(* Logix 5000 project; controller cal1632 1756-L62 rev 16.20; software revision 16.05; part 28 of 61 *)
(* tags used below, declared in another part *)
   FAULT : BOOL;
   HMI : BOOL;
   p01_recipe_active : recipe;
   p01r09_pb_global_reset : BOOL;
   p02_dint_from_hmi : hmi_dint;
   p02_real_from_hmi : hmi_real;
   p20_ai_lc01 : REAL;
   p20_di_clutch_prs_ok : BOOL;
   p20_di_loa_active : BOOL;
   p20_di_loa_fwd_dir : BOOL;
   p20_di_lob_fwd_dir : BOOL;
   p20_dint_to_hmi : DINT[16];
   p20_param_high_ki : REAL;
   p20_param_high_kp : REAL;
   p20_param_high_upd : REAL;
   p20r07 : routine;
   p20r07_timer_fault : TIMER[4];
   p20r07_timer_warning : TIMER[4];
   p20r08 : routine;
   p20r08_timer_fault : TIMER[4];
   p20r08_timer_warning : TIMER[4];
   p20r09 : routine;
   p20r09_acc_toggle : SYS_Toggle;
   p20r09_accumulator_auto : BOOL;
   p20r09_letoff_a_active : BOOL;
   p20r09_timer_fault : TIMER[4];
   p20r09_timer_warning : TIMER[4];
   p20r10 : routine;
   p20r10_param_acc_full_psn : REAL;
   p20r10_param_fill_gain : REAL;
   p20r10_param_normal_gain : REAL;
   p20r10_param_psn_gain : REAL;
   p20r10_pid_psn : PID;
   p20r10_pid_psn_cv : REAL;
   p20r10_pid_psn_pv : REAL;
   p20r10_pid_tens : PID;
   p20r10_pid_tens_cv : REAL;
   p20r10_pid_tens_pv : REAL;
   p20r10_run_permissive : BOOL;
   p20r10_speed_offset : REAL;
   p20r10_speed_offset_psn : REAL;
   p20r10_speed_offset_tens : REAL;
   p20r10_tension_request : BOOL;
   p20r10_timer : TIMER[2];
   p20r10_timer_fault : TIMER[4];
   p20r10_timer_warning : TIMER[4];
   p20r13_ai_acc_pct : REAL;
   p20r13_state : DINT;
   p20r15 : routine;
   p20r15_request_tension : BOOL;
   p20r15_request_thread_fwd : BOOL;
   p20r15_request_thread_rev : BOOL;
   p20r16 : routine;
   p20r16_request_tension : BOOL;
   p20r16_request_thread_fwd : BOOL;
   p20r16_request_thread_rev : BOOL;
   p20r18 : routine;
(* P20_Letoff, continued *)

ROUTINE R07_Alarms   (* ladder *)
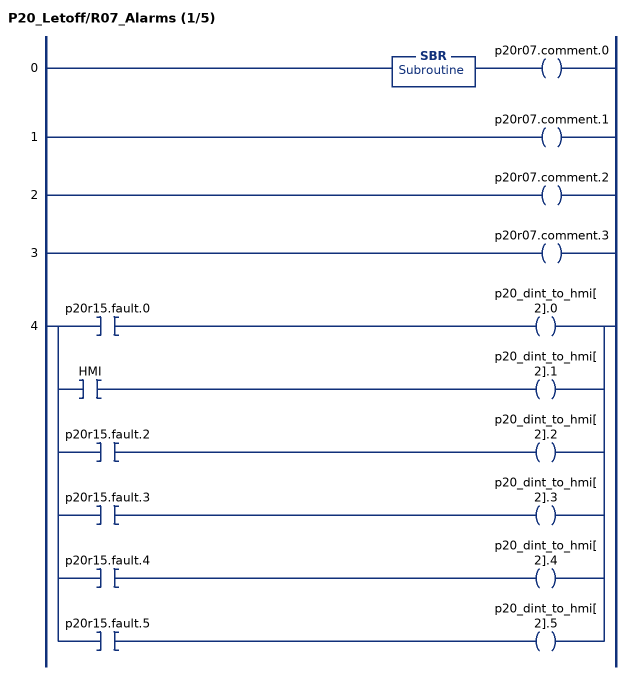
   0: SBR()OTE(p20r07.comment.0);
   1: OTE(p20r07.comment.1);
   2: OTE(p20r07.comment.2);
   3: OTE(p20r07.comment.3);
   4: [XIC(p20r15.fault.0) OTE(p20_dint_to_hmi[2].0) ,XIC(HMI) OTE(p20_dint_to_hmi[2].1) ,XIC(p20r15.fault.2) OTE(p20_dint_to_hmi[2].2) ,XIC(p20r15.fault.3) OTE(p20_dint_to_hmi[2].3) ,XIC(p20r15.fault.4) OTE(p20_dint_to_hmi[2].4) ,XIC(p20r15.fault.5) OTE(p20_dint_to_hmi[2].5) ];
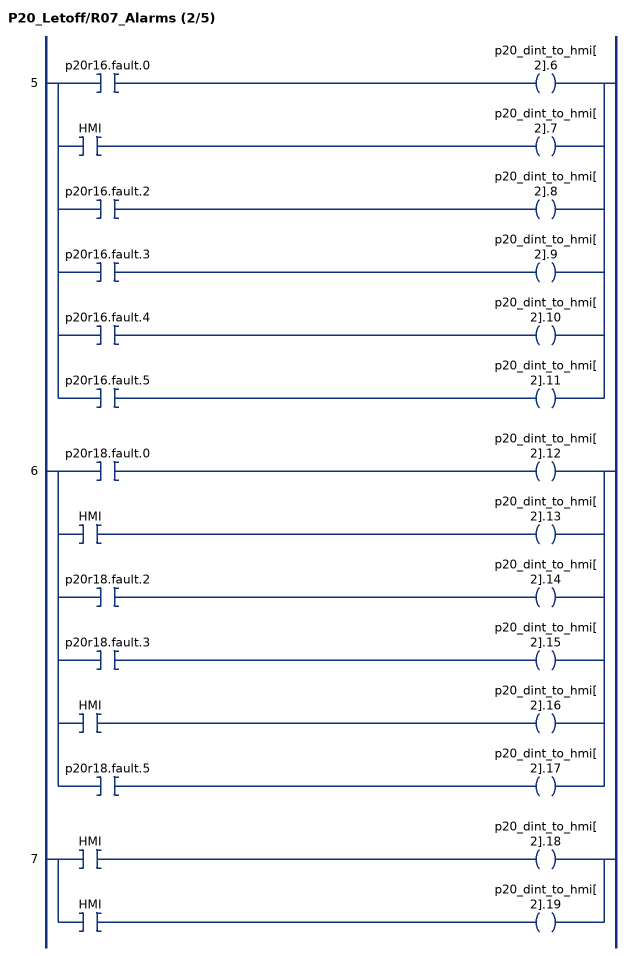
   5: [XIC(p20r16.fault.0) OTE(p20_dint_to_hmi[2].6) ,XIC(HMI) OTE(p20_dint_to_hmi[2].7) ,XIC(p20r16.fault.2) OTE(p20_dint_to_hmi[2].8) ,XIC(p20r16.fault.3) OTE(p20_dint_to_hmi[2].9) ,XIC(p20r16.fault.4) OTE(p20_dint_to_hmi[2].10) ,XIC(p20r16.fault.5) OTE(p20_dint_to_hmi[2].11) ];
   6: [XIC(p20r18.fault.0) OTE(p20_dint_to_hmi[2].12) ,XIC(HMI) OTE(p20_dint_to_hmi[2].13) ,XIC(p20r18.fault.2) OTE(p20_dint_to_hmi[2].14) ,XIC(p20r18.fault.3) OTE(p20_dint_to_hmi[2].15) ,XIC(HMI) OTE(p20_dint_to_hmi[2].16) ,XIC(p20r18.fault.5) OTE(p20_dint_to_hmi[2].17) ];
   7: [XIC(HMI) OTE(p20_dint_to_hmi[2].18) ,XIC(HMI) OTE(p20_dint_to_hmi[2].19) ];
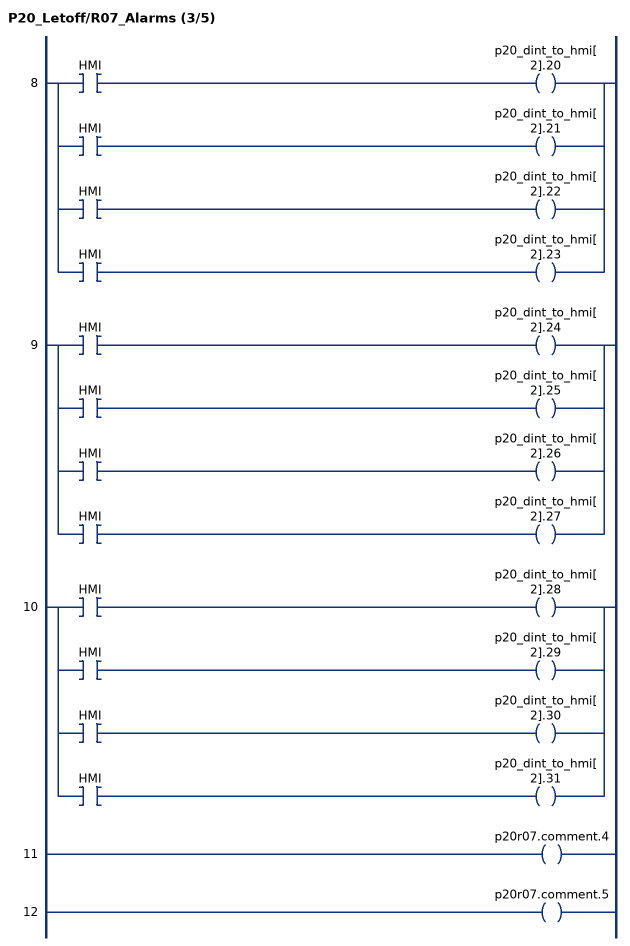
   8: [XIC(HMI) OTE(p20_dint_to_hmi[2].20) ,XIC(HMI) OTE(p20_dint_to_hmi[2].21) ,XIC(HMI) OTE(p20_dint_to_hmi[2].22) ,XIC(HMI) OTE(p20_dint_to_hmi[2].23) ];
   9: [XIC(HMI) OTE(p20_dint_to_hmi[2].24) ,XIC(HMI) OTE(p20_dint_to_hmi[2].25) ,XIC(HMI) OTE(p20_dint_to_hmi[2].26) ,XIC(HMI) OTE(p20_dint_to_hmi[2].27) ];
   10: [XIC(HMI) OTE(p20_dint_to_hmi[2].28) ,XIC(HMI) OTE(p20_dint_to_hmi[2].29) ,XIC(HMI) OTE(p20_dint_to_hmi[2].30) ,XIC(HMI) OTE(p20_dint_to_hmi[2].31) ];
   11: OTE(p20r07.comment.4);
   12: OTE(p20r07.comment.5);
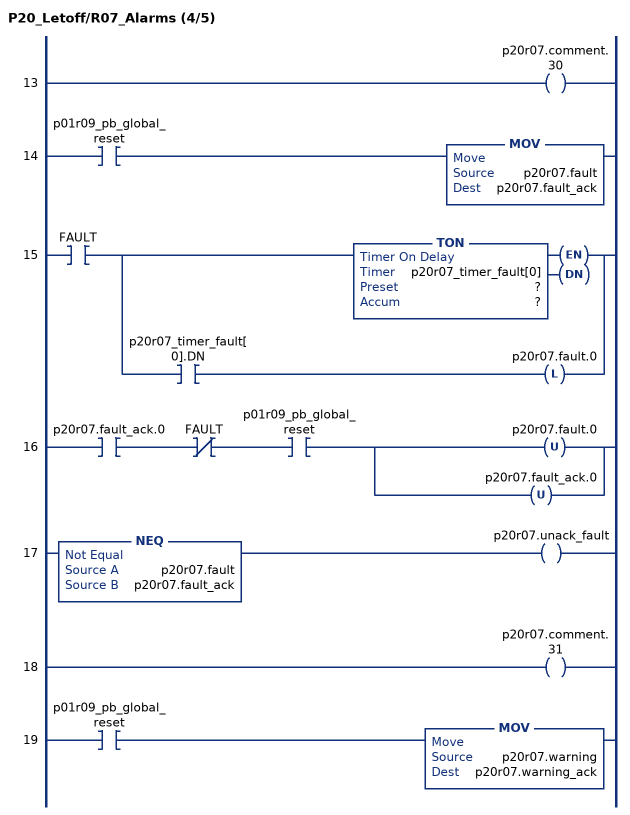
   13: OTE(p20r07.comment.30);
   14: XIC(p01r09_pb_global_reset)MOV(p20r07.fault,p20r07.fault_ack);
   15: XIC(FAULT)[TON(p20r07_timer_fault[0],?,?) ,XIC(p20r07_timer_fault[0].DN) OTL(p20r07.fault.0) ];
   16: XIC(p20r07.fault_ack.0)XIO(FAULT)XIC(p01r09_pb_global_reset)[OTU(p20r07.fault.0) ,OTU(p20r07.fault_ack.0) ];
   17: NEQ(p20r07.fault,p20r07.fault_ack)OTE(p20r07.unack_fault);
   18: OTE(p20r07.comment.31);
   19: XIC(p01r09_pb_global_reset)MOV(p20r07.warning,p20r07.warning_ack);
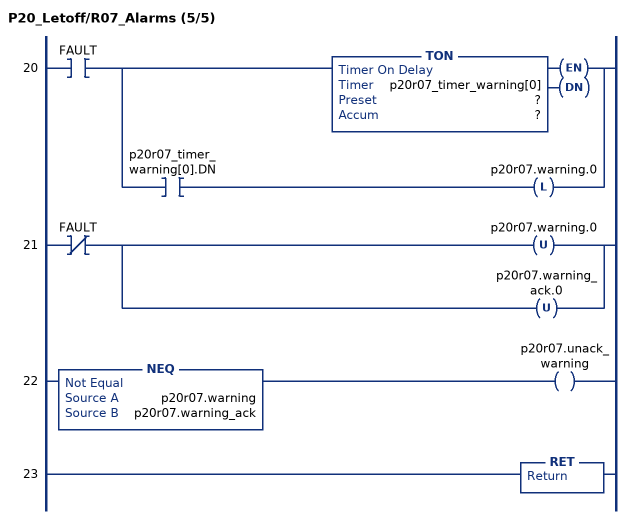
   20: XIC(FAULT)[TON(p20r07_timer_warning[0],?,?) ,XIC(p20r07_timer_warning[0].DN) OTL(p20r07.warning.0) ];
   21: XIO(FAULT)[OTU(p20r07.warning.0) ,OTU(p20r07.warning_ack.0) ];
   22: NEQ(p20r07.warning,p20r07.warning_ack)OTE(p20r07.unack_warning);
   23: RET();
END_ROUTINE

ROUTINE R08_Warnings   (* ladder *)
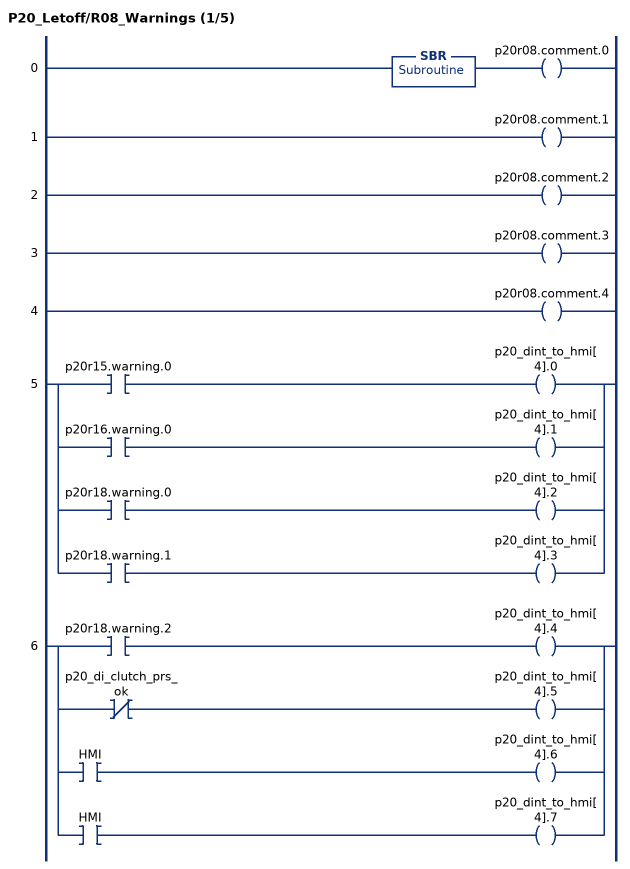
   0: SBR()OTE(p20r08.comment.0);
   1: OTE(p20r08.comment.1);
   2: OTE(p20r08.comment.2);
   3: OTE(p20r08.comment.3);
   4: OTE(p20r08.comment.4);
   5: [XIC(p20r15.warning.0) OTE(p20_dint_to_hmi[4].0) ,XIC(p20r16.warning.0) OTE(p20_dint_to_hmi[4].1) ,XIC(p20r18.warning.0) OTE(p20_dint_to_hmi[4].2) ,XIC(p20r18.warning.1) OTE(p20_dint_to_hmi[4].3) ];
   6: [XIC(p20r18.warning.2) OTE(p20_dint_to_hmi[4].4) ,XIO(p20_di_clutch_prs_ok) OTE(p20_dint_to_hmi[4].5) ,XIC(HMI) OTE(p20_dint_to_hmi[4].6) ,XIC(HMI) OTE(p20_dint_to_hmi[4].7) ];
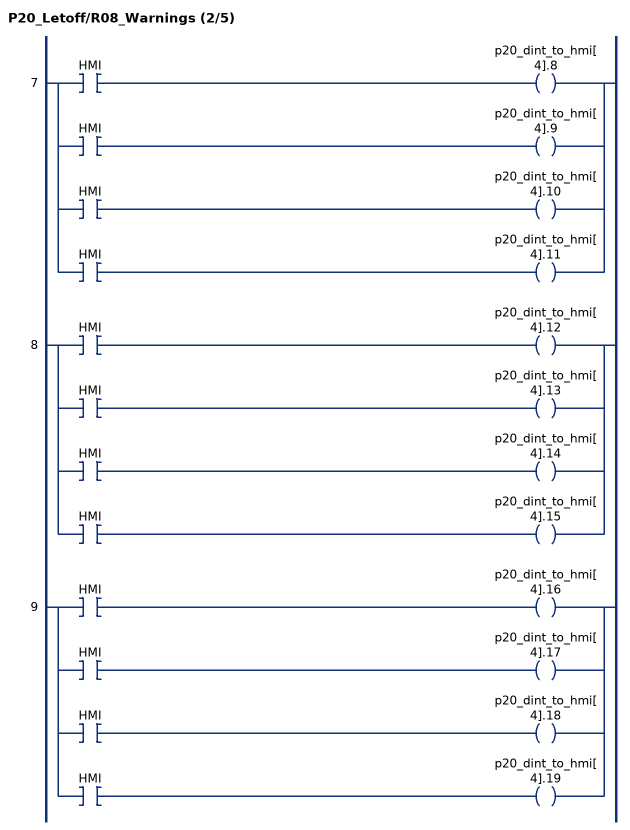
   7: [XIC(HMI) OTE(p20_dint_to_hmi[4].8) ,XIC(HMI) OTE(p20_dint_to_hmi[4].9) ,XIC(HMI) OTE(p20_dint_to_hmi[4].10) ,XIC(HMI) OTE(p20_dint_to_hmi[4].11) ];
   8: [XIC(HMI) OTE(p20_dint_to_hmi[4].12) ,XIC(HMI) OTE(p20_dint_to_hmi[4].13) ,XIC(HMI) OTE(p20_dint_to_hmi[4].14) ,XIC(HMI) OTE(p20_dint_to_hmi[4].15) ];
   9: [XIC(HMI) OTE(p20_dint_to_hmi[4].16) ,XIC(HMI) OTE(p20_dint_to_hmi[4].17) ,XIC(HMI) OTE(p20_dint_to_hmi[4].18) ,XIC(HMI) OTE(p20_dint_to_hmi[4].19) ];
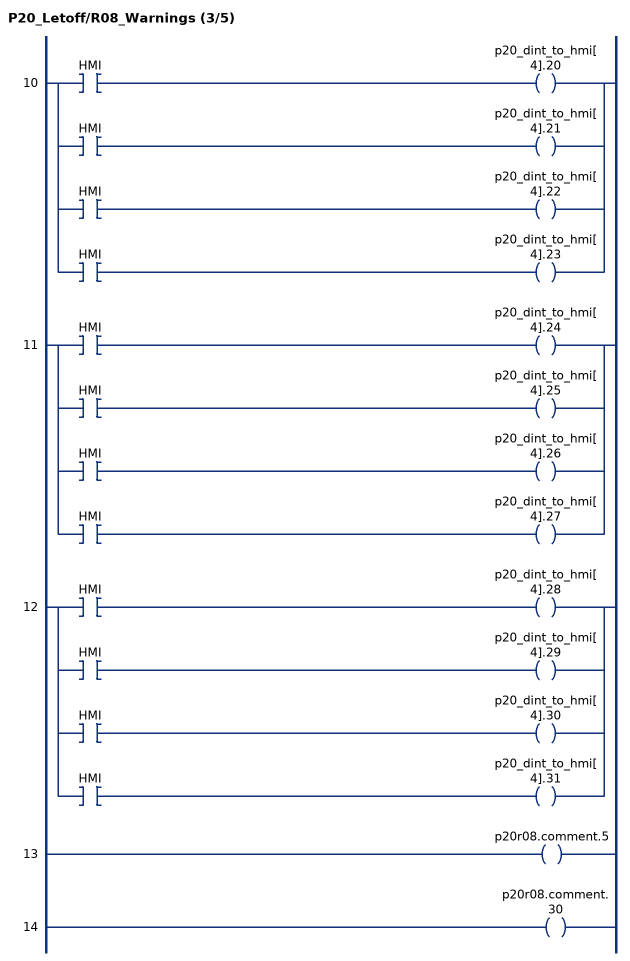
   10: [XIC(HMI) OTE(p20_dint_to_hmi[4].20) ,XIC(HMI) OTE(p20_dint_to_hmi[4].21) ,XIC(HMI) OTE(p20_dint_to_hmi[4].22) ,XIC(HMI) OTE(p20_dint_to_hmi[4].23) ];
   11: [XIC(HMI) OTE(p20_dint_to_hmi[4].24) ,XIC(HMI) OTE(p20_dint_to_hmi[4].25) ,XIC(HMI) OTE(p20_dint_to_hmi[4].26) ,XIC(HMI) OTE(p20_dint_to_hmi[4].27) ];
   12: [XIC(HMI) OTE(p20_dint_to_hmi[4].28) ,XIC(HMI) OTE(p20_dint_to_hmi[4].29) ,XIC(HMI) OTE(p20_dint_to_hmi[4].30) ,XIC(HMI) OTE(p20_dint_to_hmi[4].31) ];
   13: OTE(p20r08.comment.5);
   14: OTE(p20r08.comment.30);
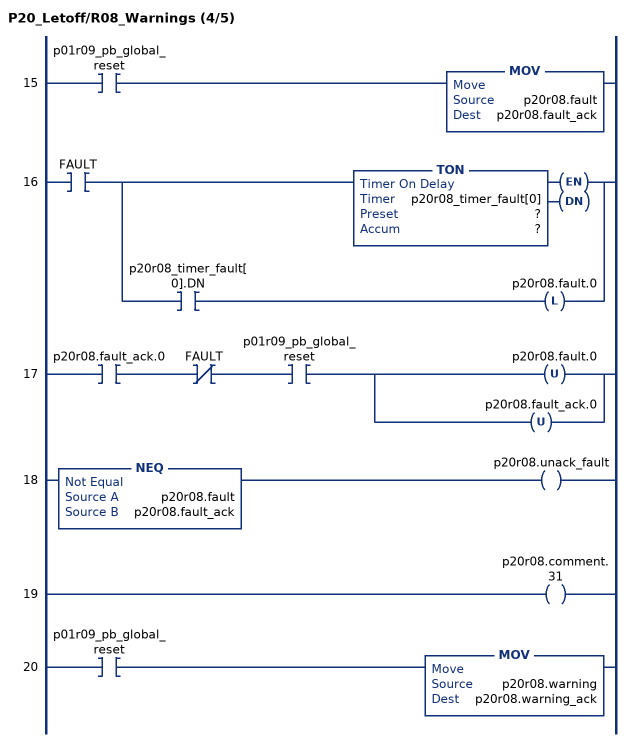
   15: XIC(p01r09_pb_global_reset)MOV(p20r08.fault,p20r08.fault_ack);
   16: XIC(FAULT)[TON(p20r08_timer_fault[0],?,?) ,XIC(p20r08_timer_fault[0].DN) OTL(p20r08.fault.0) ];
   17: XIC(p20r08.fault_ack.0)XIO(FAULT)XIC(p01r09_pb_global_reset)[OTU(p20r08.fault.0) ,OTU(p20r08.fault_ack.0) ];
   18: NEQ(p20r08.fault,p20r08.fault_ack)OTE(p20r08.unack_fault);
   19: OTE(p20r08.comment.31);
   20: XIC(p01r09_pb_global_reset)MOV(p20r08.warning,p20r08.warning_ack);
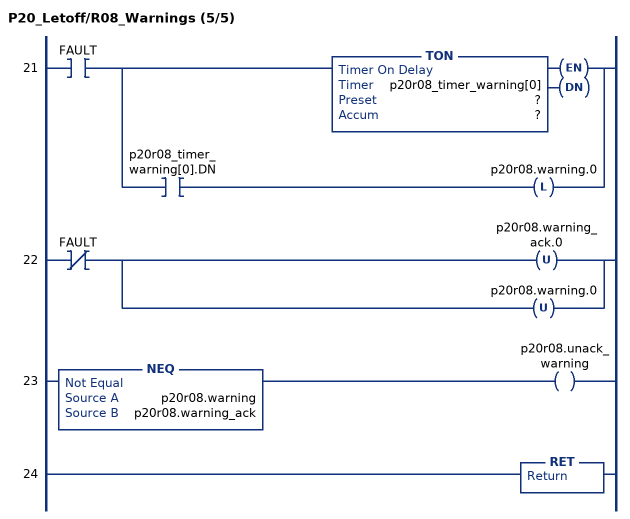
   21: XIC(FAULT)[TON(p20r08_timer_warning[0],?,?) ,XIC(p20r08_timer_warning[0].DN) OTL(p20r08.warning.0) ];
   22: XIO(FAULT)[OTU(p20r08.warning_ack.0) ,OTU(p20r08.warning.0) ];
   23: NEQ(p20r08.warning,p20r08.warning_ack)OTE(p20r08.unack_warning);
   24: RET();
END_ROUTINE

ROUTINE R09_Modes   (* ladder *)
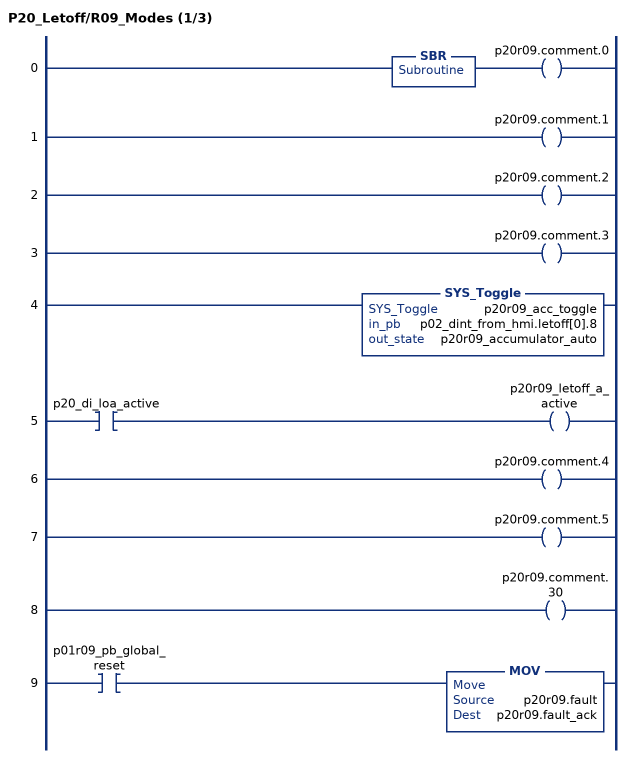
   0: SBR()OTE(p20r09.comment.0);
   1: OTE(p20r09.comment.1);
   2: OTE(p20r09.comment.2);
   3: OTE(p20r09.comment.3);
   4: SYS_Toggle(p20r09_acc_toggle,p02_dint_from_hmi.letoff[0].8,p20r09_accumulator_auto);
   5: XIC(p20_di_loa_active)OTE(p20r09_letoff_a_active);
   6: OTE(p20r09.comment.4);
   7: OTE(p20r09.comment.5);
   8: OTE(p20r09.comment.30);
   9: XIC(p01r09_pb_global_reset)MOV(p20r09.fault,p20r09.fault_ack);
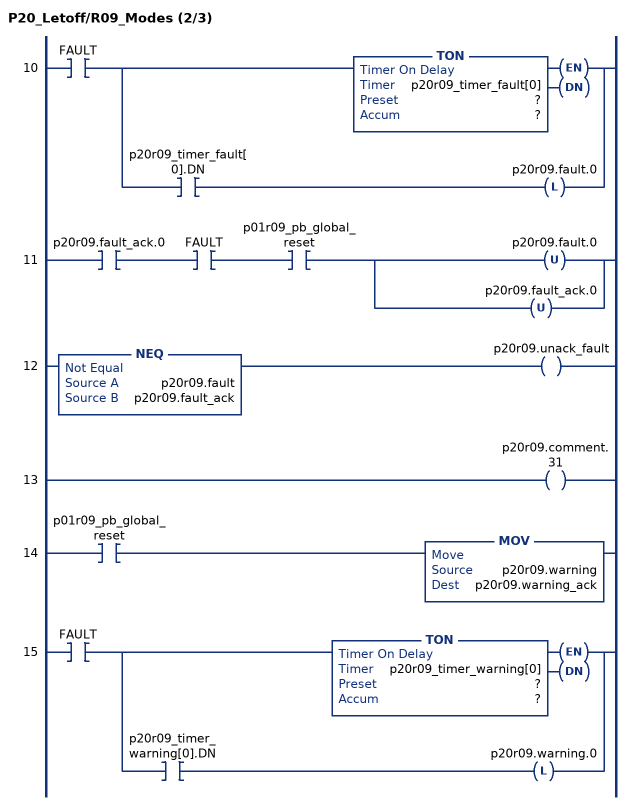
   10: XIC(FAULT)[TON(p20r09_timer_fault[0],?,?) ,XIC(p20r09_timer_fault[0].DN) OTL(p20r09.fault.0) ];
   11: XIC(p20r09.fault_ack.0)XIC(FAULT)XIC(p01r09_pb_global_reset)[OTU(p20r09.fault.0) ,OTU(p20r09.fault_ack.0) ];
   12: NEQ(p20r09.fault,p20r09.fault_ack)OTE(p20r09.unack_fault);
   13: OTE(p20r09.comment.31);
   14: XIC(p01r09_pb_global_reset)MOV(p20r09.warning,p20r09.warning_ack);
   15: XIC(FAULT)[TON(p20r09_timer_warning[0],?,?) ,XIC(p20r09_timer_warning[0].DN) OTL(p20r09.warning.0) ];
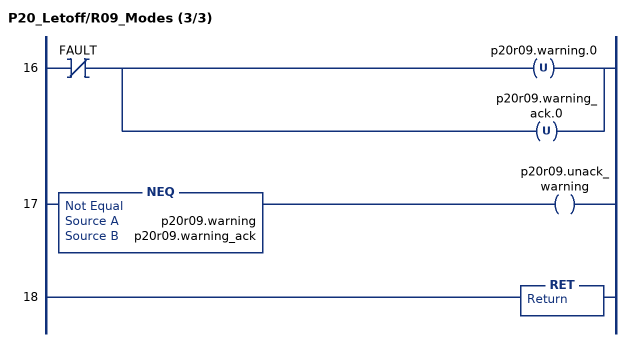
   16: XIO(FAULT)[OTU(p20r09.warning.0) ,OTU(p20r09.warning_ack.0) ];
   17: NEQ(p20r09.warning,p20r09.warning_ack)OTE(p20r09.unack_warning);
   18: RET();
END_ROUTINE

ROUTINE R10_Letoff_Speed_Control   (* ladder *)
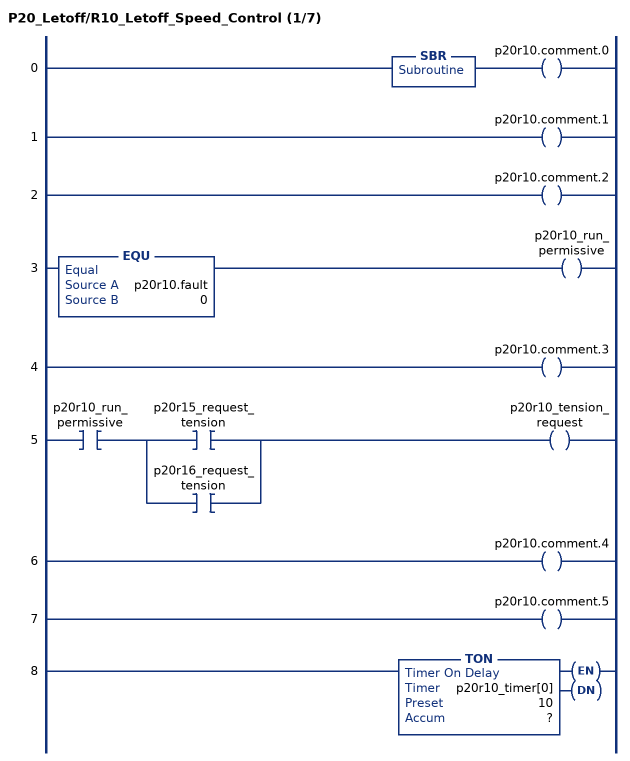
   0: SBR()OTE(p20r10.comment.0);
   1: OTE(p20r10.comment.1);
   2: OTE(p20r10.comment.2);
   3: EQU(p20r10.fault,0)OTE(p20r10_run_permissive);
   4: OTE(p20r10.comment.3);
   5: XIC(p20r10_run_permissive)[XIC(p20r15_request_tension) ,XIC(p20r16_request_tension) ]OTE(p20r10_tension_request);
   6: OTE(p20r10.comment.4);
   7: OTE(p20r10.comment.5);
   8: TON(p20r10_timer[0],?,?);
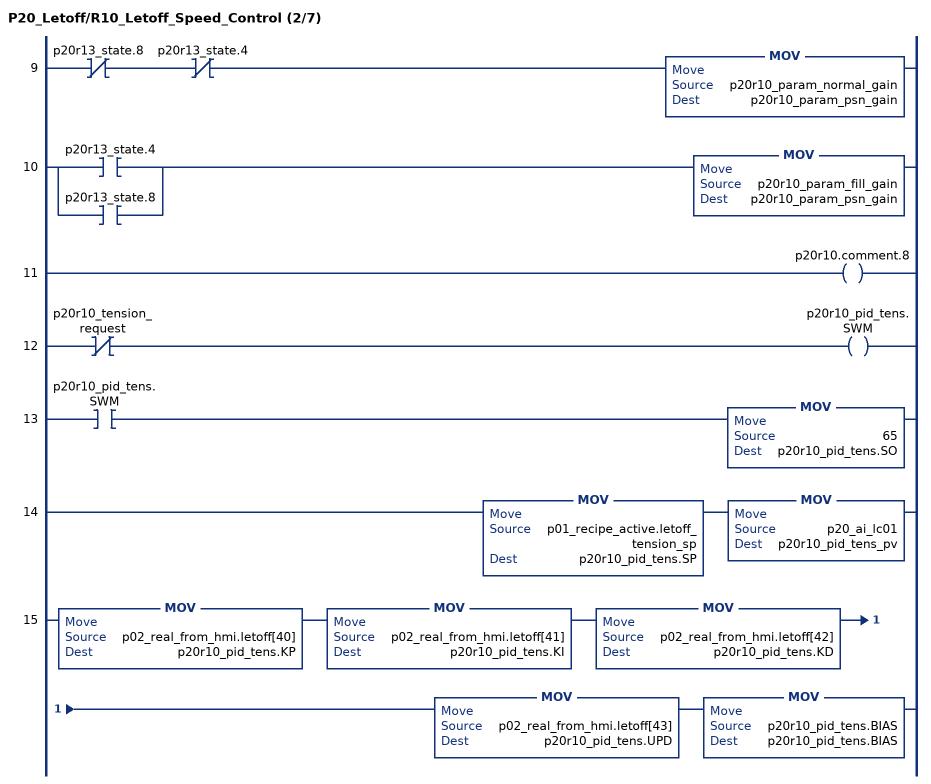
   9: XIO(p20r13_state.8)XIO(p20r13_state.4)MOV(p20r10_param_normal_gain,p20r10_param_psn_gain);
   10: [XIC(p20r13_state.4) ,XIC(p20r13_state.8) ]MOV(p20r10_param_fill_gain,p20r10_param_psn_gain);
   11: OTE(p20r10.comment.8);
   12: XIO(p20r10_tension_request)OTE(p20r10_pid_tens.SWM);
   13: XIC(p20r10_pid_tens.SWM)MOV(65,p20r10_pid_tens.SO);
   14: MOV(p01_recipe_active.letoff_tension_sp,p20r10_pid_tens.SP)MOV(p20_ai_lc01,p20r10_pid_tens_pv);
   15: MOV(p02_real_from_hmi.letoff[40],p20r10_pid_tens.KP)MOV(p02_real_from_hmi.letoff[41],p20r10_pid_tens.KI)MOV(p02_real_from_hmi.letoff[42],p20r10_pid_tens.KD)MOV(p02_real_from_hmi.letoff[43],p20r10_pid_tens.UPD)MOV(p20r10_pid_tens.BIAS,p20r10_pid_tens.BIAS);
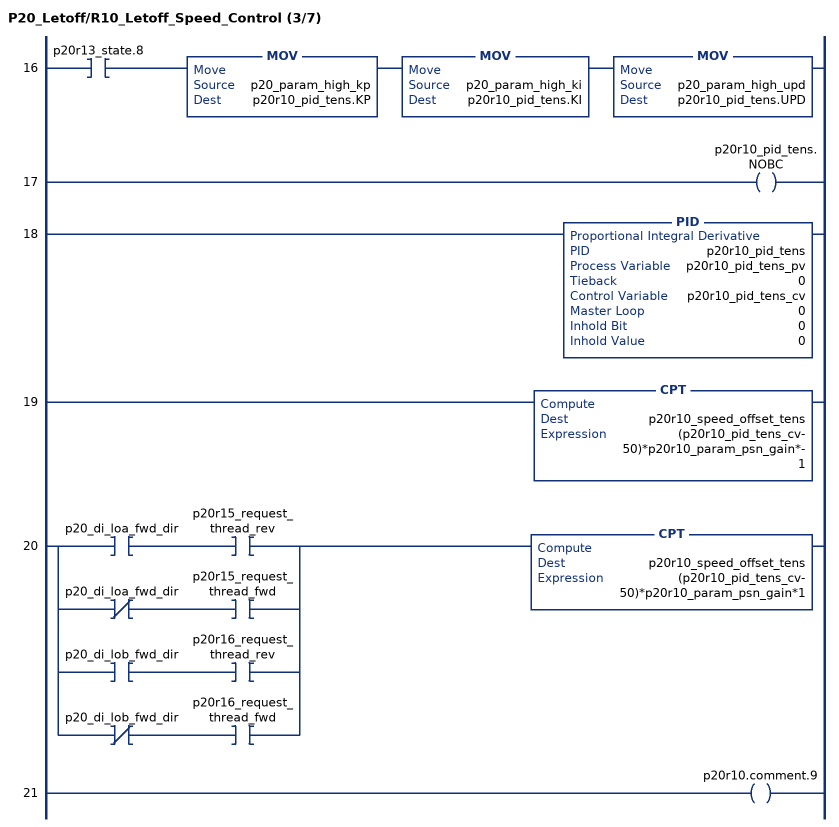
   16: XIC(p20r13_state.8)MOV(p20_param_high_kp,p20r10_pid_tens.KP)MOV(p20_param_high_ki,p20r10_pid_tens.KI)MOV(p20_param_high_upd,p20r10_pid_tens.UPD);
   17: OTE(p20r10_pid_tens.NOBC);
   18: PID(p20r10_pid_tens,p20r10_pid_tens_pv,0,p20r10_pid_tens_cv,0,0,0);
   19: CPT(p20r10_speed_offset_tens,(p20r10_pid_tens_cv-50)*p20r10_param_psn_gain*-1);
   20: [XIC(p20_di_loa_fwd_dir) XIC(p20r15_request_thread_rev) ,XIO(p20_di_loa_fwd_dir) XIC(p20r15_request_thread_fwd) ,XIC(p20_di_lob_fwd_dir) XIC(p20r16_request_thread_rev) ,XIO(p20_di_lob_fwd_dir) XIC(p20r16_request_thread_fwd) ]CPT(p20r10_speed_offset_tens,(p20r10_pid_tens_cv-50)*p20r10_param_psn_gain*1);
   21: OTE(p20r10.comment.9);
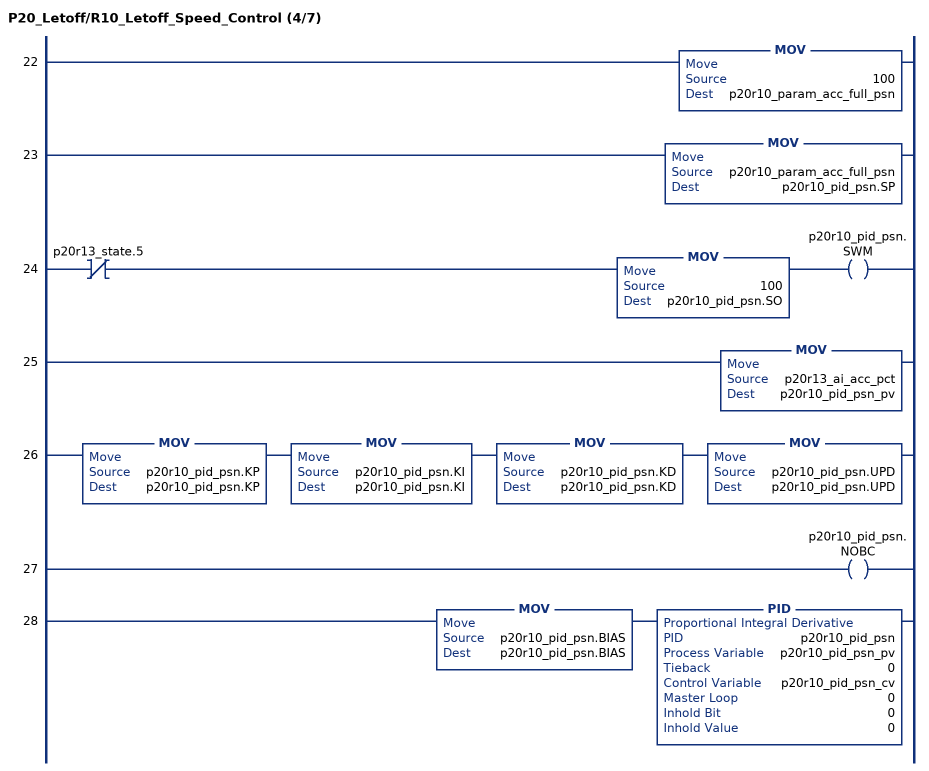
   22: MOV(100,p20r10_param_acc_full_psn);
   23: MOV(p20r10_param_acc_full_psn,p20r10_pid_psn.SP);
   24: XIO(p20r13_state.5)MOV(100,p20r10_pid_psn.SO)OTE(p20r10_pid_psn.SWM);
   25: MOV(p20r13_ai_acc_pct,p20r10_pid_psn_pv);
   26: MOV(p20r10_pid_psn.KP,p20r10_pid_psn.KP)MOV(p20r10_pid_psn.KI,p20r10_pid_psn.KI)MOV(p20r10_pid_psn.KD,p20r10_pid_psn.KD)MOV(p20r10_pid_psn.UPD,p20r10_pid_psn.UPD);
   27: OTE(p20r10_pid_psn.NOBC);
   28: MOV(p20r10_pid_psn.BIAS,p20r10_pid_psn.BIAS)PID(p20r10_pid_psn,p20r10_pid_psn_pv,0,p20r10_pid_psn_cv,0,0,0);
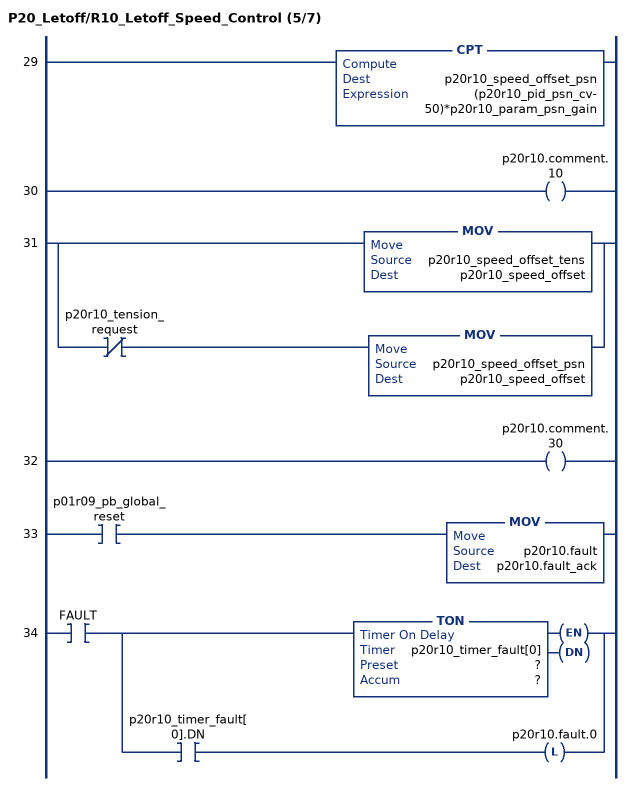
   29: CPT(p20r10_speed_offset_psn,(p20r10_pid_psn_cv-50)*p20r10_param_psn_gain);
   30: OTE(p20r10.comment.10);
   31: [MOV(p20r10_speed_offset_tens,p20r10_speed_offset) ,XIO(p20r10_tension_request) MOV(p20r10_speed_offset_psn,p20r10_speed_offset) ];
   32: OTE(p20r10.comment.30);
   33: XIC(p01r09_pb_global_reset)MOV(p20r10.fault,p20r10.fault_ack);
   34: XIC(FAULT)[TON(p20r10_timer_fault[0],?,?) ,XIC(p20r10_timer_fault[0].DN) OTL(p20r10.fault.0) ];
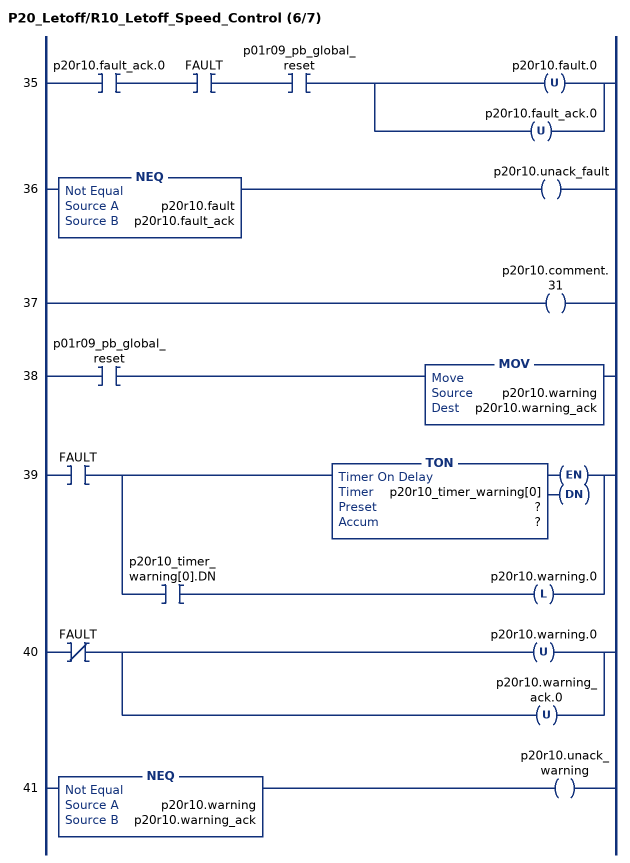
   35: XIC(p20r10.fault_ack.0)XIC(FAULT)XIC(p01r09_pb_global_reset)[OTU(p20r10.fault.0) ,OTU(p20r10.fault_ack.0) ];
   36: NEQ(p20r10.fault,p20r10.fault_ack)OTE(p20r10.unack_fault);
   37: OTE(p20r10.comment.31);
   38: XIC(p01r09_pb_global_reset)MOV(p20r10.warning,p20r10.warning_ack);
   39: XIC(FAULT)[TON(p20r10_timer_warning[0],?,?) ,XIC(p20r10_timer_warning[0].DN) OTL(p20r10.warning.0) ];
   40: XIO(FAULT)[OTU(p20r10.warning.0) ,OTU(p20r10.warning_ack.0) ];
   41: NEQ(p20r10.warning,p20r10.warning_ack)OTE(p20r10.unack_warning);
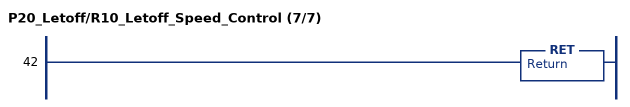
   42: RET();
END_ROUTINE
